// SIMATIC STEP 7 (V5.x) project GRAFCET
// CPU: CPU313 C-2 DP(1)
// station: P_ADR_BUS
// station: Hardware
// station: SIMATIC 300 Station

SYMBOL_TABLE
"G7_STD_3"	FC 72	FC 72
"Stop Btn"	I 0.0	BOOL	// Stop the motor
"Start Btn Direct"	I 0.1	BOOL	// Button input direct direction
"Start Btn Inverse"	I 0.2	BOOL	// Button input inverse direction
"Cycle Execution"	OB 1	OB 1
"KM Direct"	Q 0.0	BOOL	// Drive the motor in the direct direction
"KM Inverse"	Q 0.1	BOOL	// Drive the motor in the inverse direction
"TIME_TCK"	SFC 64	SFC 64	// Read the System Time
END_SYMBOL_TABLE
